(* IEC 61131-3 sources: Lasal/CPU_5344_V01/Class/checkClampOk, 1 file *)

(* ---- checkClampOk.st ---- *)
(*!
<Class
	Name               = "checkClampOk"
	Revision           = "0.0"
	RealtimeTask       = "false"
	CyclicTask         = "false"
	BackgroundTask     = "false"
	Sigmatek           = "false"
	OSInterface        = "false"
	HighPriority       = "false"
	Automatic          = "false"
	UpdateMode         = "Prescan"
	SharedCommandTable = "true"
	Objectsize         = "(284,120)">
	<Channels>
		<Server Name="ClassSvr" Visualized="false" Initialize="false" WriteProtected="true" Retentive="false"/>
		<Client Name="iActState" Required="true" Internal="false"/>
		<Client Name="sShouldBeState" Required="true" Internal="false"/>
	</Channels>
</Class>
*)
checkClampOk : CLASS
  //Servers:
	ClassSvr 	: SvrChCmd_DINT;
  //Clients:
	iActState 	: CltCh_cilPos;
	sShouldBeState 	: CltCh_cilPos;
  //Variables:
  //Functions:

	FUNCTION VIRTUAL GLOBAL ClassSvr::Read
		VAR_OUTPUT
			output (EAX) 	: DINT;
		END_VAR;
  //Tables:
	FUNCTION @STD
		VAR_OUTPUT
			ret_code	: CONFSTATES;
		END_VAR;
	FUNCTION GLOBAL TAB @CT_;
END_CLASS;

// JdK 12-6-2019 created for Traffiroad 4284/standard lib
// simple class to check if a cilinder is in the state it should be te be ok

FUNCTION VIRTUAL GLOBAL checkClampOk::ClassSvr::Read
	VAR_OUTPUT
		output (EAX) 	: DINT;
	END_VAR

  iActState:=iActState.Read();
  sShouldBeState:=sShouldBeState.Read();

  IF iActState=sShouldBeState THEN
    ClassSvr:=1;
  ELSE
    ClassSvr:=0;
  END_IF;

	output := ClassSvr;

END_FUNCTION
